INTERFACE I_Property EXTENDS __SYSTEM.IQueryInterface, I_Disposable, I_DataAccess

METHOD PUBLIC Accept
VAR_INPUT
	Visitor : I_PropertyVisitor;
END_VAR
END_METHOD

METHOD PUBLIC Configure
VAR_INPUT
	Settings : I_PropertySettings;
END_VAR
END_METHOD

PROPERTY PUBLIC Name : T_MAXSTRING
GET
END_GET
END_PROPERTY

END_INTERFACE

(* stored: Version 1.1.0.1, ProductVersion 3.1.4024.12
   Itf I_Property: Id {01df4a8d-eb1b-0f3a-1311-1bc4ca42d2d5}
   Method Accept: Id {2833095d-c1ba-073d-2fe5-a4ab2f0685a6}
   Method Configure: Id {a5a48b39-2a3b-0b94-0b40-72d07ea41510}
   Property Name: Id {c64e0aa6-0931-0bc7-1c4c-2bf3f1baaa60}
   Get Get: Id {a5aa0fd1-8b9e-0fa9-2e9f-5d84bf9eb18e} *)
